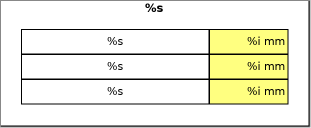
VISUALIZATION VISU_CONFIG_POSITION_REF  // 311x128
VAR_IN_OUT
	m_Input_Index:			INT;
END_VAR
    RoundedRectangle (0,0 309x126), "%s", text list: 'TextList_Config_Mouvements', text index: 2
    Rectangle (209,29 79x25), "%i mm", text variable: PRG_MOUVEMENT_PS.PRM_POS_REF[m_Input_Index,1], input disabled if: NOT Global_Variables.PRG_USER.ACTU_USER.CONF_MACHINE
        OnMouseDown: write the text variable via VisuDialogs.Numpad, min 0, max 900
    Rectangle (21,29 188x25), "%s", text list: 'TextList_Position_Canne', text index: 1
    Rectangle (21,54 188x25), "%s", text list: 'TextList_Position_Canne', text index: 2
    Rectangle (21,79 188x25), "%s", text list: 'TextList_Position_Canne', text index: 3
    Rectangle (209,54 79x25), "%i mm", text variable: PRG_MOUVEMENT_PS.PRM_POS_REF[m_Input_Index,2], input disabled if: NOT Global_Variables.PRG_USER.ACTU_USER.CONF_MACHINE
        OnMouseDown: write the text variable via VisuDialogs.Numpad, min 0, max 900
    Rectangle (209,79 79x25), "%i mm", text variable: PRG_MOUVEMENT_PS.PRM_POS_REF[m_Input_Index,3], input disabled if: NOT Global_Variables.PRG_USER.ACTU_USER.CONF_MACHINE
        OnMouseDown: write the text variable via VisuDialogs.Numpad, min 0, max 900
END_VISUALIZATION

(* stored: Version 1.1.0.1, ProductVersion 3.1.4024.10
   Visu VISU_CONFIG_POSITION_REF: Id {76c301a3-634d-41c5-bd2e-e0d541c7b726} *)
